// TwinCAT 3 PLC project PLC01
// ProgramVersion: 3.1.4023.0
// libraries:
//   Tc2_Standard, * (Beckhoff Automation GmbH)
//   Tc2_System, * (Beckhoff Automation GmbH)
//   Tc2_Utilities, * (Beckhoff Automation GmbH)
//   Tc3_Module, * (Beckhoff Automation GmbH)
// project tree:
//   DUTs/ stAlarmHist.TcDUT
//   / GlobalTextList.TcGTLO, PlcTask.TcTTO, Visualization Manager.TcVMO (not stored)
//   GVLs/ fromHMI.TcGVL, toHMI.TcGVL
//   POUs/ FB_AlarmHistCtrl.TcPOU, MAIN.TcPOU, prgAlarms.TcPOU
//   VISUs/ alarmHist.TcVIS, Visualization.TcVIS
// real-time tasks:
//   TASK PlcTask: cycle T#10ms, priority 20, ADS port 350

CONFIGURATION PLC01
    RESOURCE PLC ON TwinCAT3
        TASK PlcTask(INTERVAL := T#10ms, PRIORITY := 20);
        PROGRAM MAIN WITH PlcTask : MAIN;
    END_RESOURCE
END_CONFIGURATION

// ---- DUTs/stAlarmHist.TcDUT
TYPE stAlarmHist :
STRUCT
	sDate:STRING(23);
	sTime:STRING(23);
	sMessage:STRING;
END_STRUCT
END_TYPE

// ---- GVLs/fromHMI.TcGVL
{attribute 'qualified_only'}
VAR_GLOBAL
	bIhmReset:BOOL;	
END_VAR

// ---- GVLs/toHMI.TcGVL
{attribute 'qualified_only'}
VAR_GLOBAL
	aEvents:ARRAY[1..80] OF  ST_ReadEvent;
END_VAR
VAR_GLOBAL CONSTANT
	nLastHistAlarm:UINT:=50;
END_VAR
VAR_GLOBAL PERSISTENT
	aHist:ARRAY[1..nLastHistAlarm] OF stAlarmHist;			//alarm history
END_VAR

// ---- POUs/MAIN.TcPOU
PROGRAM MAIN
VAR
END_VAR

prgAlarms();

END_PROGRAM

// ---- POUs/prgAlarms.TcPOU
PROGRAM prgAlarms
VAR
	abAlarm: ARRAY[1..iNumAlarm] OF BOOL;
	aFBAlarm:ARRAY[1..iNumAlarm] OF FB_SimpleAdsLogEvent;
	i: INT;
	readEvents:FB_AdsReadEvents;
	bReadEvents: BOOL := TRUE;
	iNumEvents: UDINT;
	//Alarm Histtory
	alarmHistCtrl:FB_AlarmHistCtrl;
END_VAR
VAR CONSTANT
	iNumAlarm:INT:=54;
END_VAR

FOR i:=1 TO iNumAlarm DO
	aFBAlarm[i](
		SourceID:=1100 , 
		EventID:= i, 
		bSetEvent:= abAlarm[i], 
		bQuit:= fromHMI.bIhmReset, 
		ErrId=> , 
		Error=> );
END_FOR

readEvents(
	sNetId:= '', 
	bReadEvents:= bReadEvents, 
	nLanguageId:= 1033, 
	eDateAndTimeFormat:= E_DATEANDTIMEFORMAT.de_DE, 
	tRefreshTime:=T#1S , 
	tTimeout:=T#10S , 
	aEvents=> toHMI.aEvents, 
	nNumberOfEvents=> iNumEvents, 
	bBusy=> , 
	bDone=> , 
	bError=> , 
	nErrId=> );

alarmHistCtrl(ptHist:= ADR(toHMI.aHist), ptActiveAlarms:=ADR(toHMI.aEvents));

END_PROGRAM

// ---- POUs/FB_AlarmHistCtrl.TcPOU
FUNCTION_BLOCK FB_AlarmHistCtrl
VAR_INPUT
	ptHist:POINTER TO ARRAY[1..toHMI.nLastHistAlarm] OF stAlarmHist;			//
									//
	ptActiveAlarms:POINTER TO ARRAY[1..80] OF ST_ReadEvent;	//

END_VAR
VAR_OUTPUT
END_VAR
VAR
	nActiveAlarmOld:UDINT;	//Number of active alarms on the last cycle
	i: UDINT;
	i2:UDINT;
	bLeaveLoop: BOOL;
	bUpdateHist:BOOL;
	nCurrAlarmNum: UDINT;
	nOldAlarmNum: UDINT;
	nActiveAlarms:UDINT;
	i3: UDINT;
END_VAR
//VAR CONSTANT
//	nLastHistAlarm:UINT:=1000;
//END_VAR

nActiveAlarms:=0;
FOR i3:= 1 TO 80 DO
	IF ptActiveAlarms^[i3].nEventId <> 0 THEN
		nActiveAlarms:=i3;
	ELSE
		EXIT;	
	END_IF
END_FOR

IF nActiveAlarmOld <> nActiveAlarms AND nActiveAlarms> nActiveAlarmOld THEN
	nCurrAlarmNum:=nActiveAlarms;
	nOldAlarmNum:=nActiveAlarmOld;
	bUpdateHist:=TRUE;
END_IF

IF bUpdateHist THEN
		i:=nCurrAlarmNum;
		bLeaveLoop:=FALSE;
		WHILE NOT bLeaveLoop DO
			IF i <> nOldAlarmNum THEN
				FOR i2 := toHMI.nLastHistAlarm TO 2 BY -1 DO
					ptHist^[i2]:= ptHist^[i2-1];
				END_FOR
				ptHist^[1].sDate:=ptActiveAlarms^[i].sDate;
				ptHist^[1].sTime:=ptActiveAlarms^[i].sTime;
				ptHist^[1].sMessage:=ptActiveAlarms^[i].sMessageText;
			ELSE
				bLeaveLoop:=TRUE;
			END_IF
			i:=i-1;
		END_WHILE
	bUpdateHist:=FALSE;
END_IF

nActiveAlarmOld:=nActiveAlarms;

END_FUNCTION_BLOCK

// ---- GlobalTextList.TcGTLO
TEXTLIST GlobalTextList
  517 = 'Data'
  867 = 'Date'
  647 = 'Hora'
  205 = 'Mensagem'
  863 = 'Message'
  468 = 'Reset'
  179 = 'Time'
END_TEXTLIST

// ---- VISUs/alarmHist.TcVIS
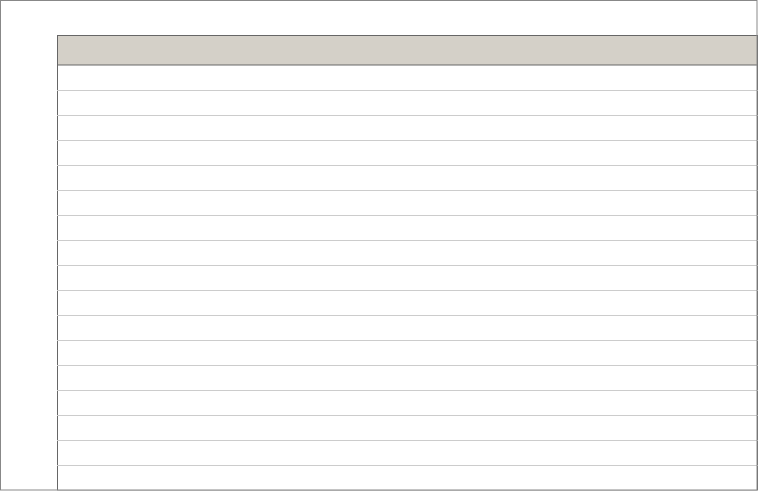
VISUALIZATION alarmHist  // 758x491
    Table (57,35 701x456), data array: toHMI.aHist
        p3854506369: toHMI.aHist[INDEX].sDate
        p1892666644: toHMI.aHist[INDEX].sTime
        p338671338: toHMI.aHist[INDEX].sMessage
END_VISUALIZATION

// ---- VISUs/Visualization.TcVIS
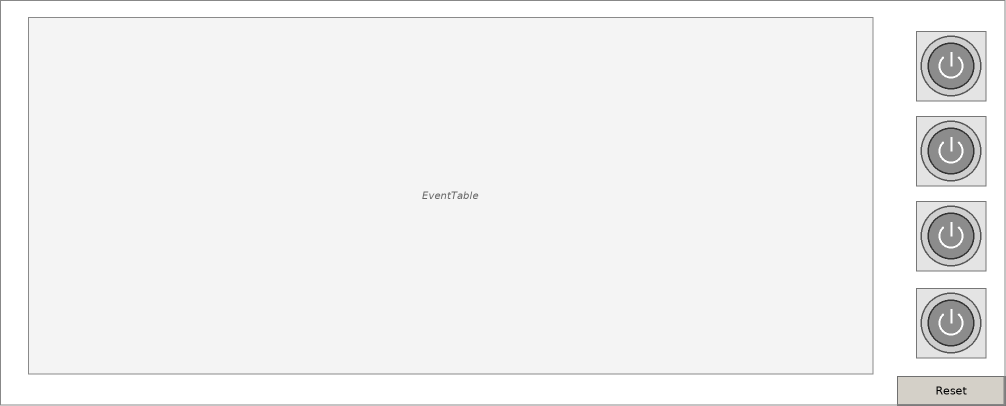
VISUALIZATION Visualization  // 1006x406
    EventTable (28,17 845x357)
        p1690906150: Class
        p3258520714: Date
        p2231227367: Time
        p3993844394: Time
        p2076579579: Details
        p3558512729: toHMI.aEvents
        p3921149237: m_pDataArray..pArray
    PowerSwitch (916,31 70x70), variable: prgAlarms.abAlarm[1], behaviour: TOGGLE, style: Switch-PowerSwitch-Gray
    PowerSwitch (916,116 70x70), variable: prgAlarms.abAlarm[2], behaviour: TOGGLE, style: Switch-PowerSwitch-Gray
    PowerSwitch (916,201 70x70), variable: prgAlarms.abAlarm[3], behaviour: TOGGLE, style: Switch-PowerSwitch-Gray
    PowerSwitch (916,288 70x70), variable: prgAlarms.abAlarm[4], behaviour: TOGGLE, style: Switch-PowerSwitch-Gray
    Button (897,376 109x30), "Reset"
        tap fromHMI.bIhmReset
END_VISUALIZATION
